(************************************************************************************************)
(*								Beckhoff Automation Poland										*)
(* 									F_Convert_4BBCD_To_Real v1.0								*)
(* 										26.06.2014												*)
(*	Funkcja konwertujaca 4 zmienne typu BYTE (BCD) na REAL - czesto spotykane w protokole M-Bus	*)
(*______________________________________________________________________________________________*)
FUNCTION F_Convert_4BBCD_To_Real : REAL
VAR_INPUT
	Byte1: BYTE; (* LSB *)
	Byte2: BYTE;
	Byte3: BYTE;
	Byte4: BYTE; (* MSB *)
END_VAR

F_Convert_4BBCD_To_Real := udint_to_real(F_BCDToDec(Byte1)*1+F_BCDToDec(Byte2)*100+F_BCDToDec(Byte3)*10000+F_BCDToDec(Byte4)*1000000);

END_FUNCTION

(* stored: Version 1.1.0.1, ProductVersion 3.1.4026.13, FileIdentifier c1ce4528486d74a1f2e3508d9d358f256b2eb694, FileSignature 37279235b8a956d89f175745fb886fcf03c16edc13f48fd03e6594759f1c1c783244997b616340ae5dd33bce024b687715a1d820d07d32685597cc844c6d6fd0d3216de0d3ce821039b3a40ea0456ebac44cb902b86638bc31d4fc8ceb1e942d2af8114c75c34229ba83d086917ace4eb8c0264f45dc22c20751b9b88b8e53d2db0349d4e02894cb9819b3a696ce1602b84c4d7508113a7dfa1f6497fa6489f3339f42cb5bc1719ed9e1eb43be5ce177d286cb99f67a5d29e0e506cd7d1a878e2b32596af9782135ecdbaab37ca64150d8e1105a2cc31c8ee30fa576ca9c35cc13b87b665b5eb7bf4830de5e83be01e4c2f3ac1c1a0dca12a50471838aedd85c
   POU F_Convert_4BBCD_To_Real: Id {2c42b93a-6c8a-4f82-91d0-b074ea38b8c7}, SpecialFunc None *)
